// TwinCAT 3 PLC project ServerSampleProject
// ProgramVersion: 3.1.0.9
// libraries:
//   Tc2_Standard, * (Beckhoff Automation GmbH)
//   Tc2_System, * (Beckhoff Automation GmbH)
//   Tc3_Interfaces, * (Beckhoff Automation GmbH)
//   Tc3_Module, * (Beckhoff Automation GmbH)
// project tree:
//   DUTs/ ST_Communication.TcDUT, ST_RecipeData.TcDUT
//   / PlcTask.TcTTO
//   POUs/ MAIN.TcPOU
// real-time tasks:
//   TASK PlcTask: cycle T#10ms, priority 20, ADS port 350

CONFIGURATION ServerSampleProject
    RESOURCE PLC ON TwinCAT3
        TASK PlcTask(INTERVAL := T#10ms, PRIORITY := 20);
        PROGRAM MAIN WITH PlcTask : MAIN;
    END_RESOURCE
END_CONFIGURATION

// ---- DUTs/ST_Communication.TcDUT
TYPE ST_Communication :
STRUCT
	Var1 : INT;
	Var2 : DINT;
	RecipeData: ST_RecipeData;
END_STRUCT
END_TYPE

// ---- DUTs/ST_RecipeData.TcDUT
TYPE ST_RecipeData :
STRUCT
	Receipt1 : INT;
	Receipt2 : INT;
END_STRUCT
END_TYPE

// ---- POUs/MAIN.TcPOU
PROGRAM MAIN
VAR
	{attribute 'OPC.UA.DA' := '1'}
	stCommunication : ST_Communication; // sample to demonstrate UA StructuredDataTypes
	{attribute 'OPC.UA.DA' := '1'}
	nCounter : INT; // sample to demonstrate UA A&C LimitAlarmType
	{attribute 'OPC.UA.DA' := '1'}
	bToogle : BOOL; // sample to demonstrate UA A&C OffNormalAlarmType 
END_VAR

END_PROGRAM
